// Block: PPrgArchive12

DATA_BLOCK PPrgArchive12
VERSION : 0.1
   NON_RETAIN
   VAR
      PRG : Array[1101..1200] of PPrg_Data;
   END_VAR

BEGIN
   // No initialization required
END_DATA_BLOCK
